FUNCTION FC_ReadJoyPos : INT
VAR_INPUT
END_VAR
VAR
END_VAR

END_FUNCTION

(* stored: Version 1.1.0.1, ProductVersion 3.1.4024.12
   POU FC_ReadJoyPos: Id {62bdda31-26e5-4b81-9425-733300eafdc1}, SpecialFunc None *)
